INTERFACE I_HE_SolidAttenuatorXRayBeamParameters EXTENDS I_Fallible


METHOD GetBeamEnergy
VAR_INPUT
    Energy : I_QuantityLREALPublic;
END_VAR
END_METHOD


METHOD GetBeamPhotonEnergy
VAR_INPUT
    PhotonEnergy : I_QuantityLREALPublic;
END_VAR
END_METHOD


METHOD GetBeamRepetitionRate
VAR_INPUT
    RepetitionRate : I_QuantityLREALPublic;
END_VAR
END_METHOD

END_INTERFACE

(* stored: Version 1.1.0.1
   Itf I_HE_SolidAttenuatorXRayBeamParameters: Id {4d048882-1b8e-4c10-be92-4b7020f1ea48}
   Method GetBeamEnergy: Id {ed2cb71e-eed3-4446-8e41-32ffe2bdb60f}
   Method GetBeamPhotonEnergy: Id {660d25f1-dff3-404e-9116-14d6d3aa9234}
   Method GetBeamRepetitionRate: Id {48c60e37-f09b-4556-a450-83975e743bda} *)
